// Implicitly generated code : DO NOT EDIT
FUNCTION CheckRangeUnsigned : UDINT
VAR_INPUT
	value, lower, upper: UDINT;
END_VAR

// Implicitly generated code : Only an Implementation suggestion
{noflow}
Fault_Count_G(CU:=FALSE) ; 
IF (value < lower) THEN
	CheckRangeUnsigned := lower;
		Fault_Count_G(CU:=TRUE) ; 
ELSIF(value > upper) THEN
	CheckRangeUnsigned := upper;
		Fault_Count_G(CU:=TRUE) ; 
ELSE
	CheckRangeUnsigned := value;
END_IF
{flow}

END_FUNCTION

(* stored: Version 1.1.0.1, ProductVersion 3.1.4024.2
   POU CheckRangeUnsigned: Id {115ceed5-0e03-4010-93f3-0c433301409f}, SpecialFunc CheckRangeUnsigned *)
